INTERFACE I_ChunkedRequestData EXTENDS I_SessionData

PROPERTY PUBLIC IsComplete : BOOL
GET
END_GET
END_PROPERTY

PROPERTY PUBLIC PayloadAddress : POINTER TO STRING
GET
END_GET
END_PROPERTY

PROPERTY PUBLIC PayloadSizeInBytes : UDINT
GET
END_GET
END_PROPERTY

METHOD PUBLIC TryAddChunkedPayload : BOOL;
VAR_INPUT
	PayloadAddress : POINTER TO STRING;
	PayloadSize : UDINT;
	ChunkSequence : DINT;
END_VAR
END_METHOD

END_INTERFACE

(* stored: Version 1.1.0.1, ProductVersion 3.1.4026.13
   Itf I_ChunkedRequestData: Id {4193533e-3ebf-4628-899a-04436528d3cb}
   Property IsComplete: Id {926f7cbd-37cd-417e-8f32-cd7262aa2b7c}
   Get Get: Id {50749355-9164-4c0f-aeeb-c4b6fbda6125}
   Property PayloadAddress: Id {a833c050-1d5a-49dc-891b-7afb4acb579d}
   Get Get: Id {430414c2-63bd-444a-a11a-eb5432a742d2}
   Property PayloadSizeInBytes: Id {cf1e60ae-357a-46b7-8ccd-95acb00a445e}
   Get Get: Id {e1212024-07dc-46fb-b103-77cc0d7c76bc}
   Method TryAddChunkedPayload: Id {350f5725-d20b-4bcd-bd5e-d226edede4bb} *)
